(* PLC project addition_10, Dassault Systèmes ControlBuild 2024x *)
(* stored: creationDateTime 2023-10-03T11:13:32-01:00 *)

(* This module simulates the addition of maximum 10 real numbers. *)
FUNCTION_BLOCK equipment_library.addition_10
  VAR_INPUT
    in1 : REAL := 0.0;
    in2 : REAL := 0.0;
    in3 : REAL := 0.0;
    in4 : REAL := 0.0;
    in5 : REAL := 0.0;
    in6 : REAL := 0.0;
    in7 : REAL := 0.0;
    in8 : REAL := 0.0;
    in9 : REAL := 0.0;
    in10 : REAL := 0.0;
  END_VAR
  VAR_OUTPUT
    realValue : REAL := 0.0;
    dintValue : DINT := 0;
    intValue : INT := 0;
  END_VAR
  VAR
    d_locking : BOOL := false;
    v_d_locking : REAL := 0.0;
  END_VAR


ACTION C_source_code:
/* ----------------------------------------------------------------	*/
/* Type : Model of Operative Behaviour					*/
/* Category :  Toolbox							*/
/* Author : Dassault Systemes						*/
/* Update date : June 2018						*/
/* ----------------------------------------------------------------	*/
/* This module simulates the addition of maximum 10 real numbers.	*/
/* réels au maximum								*/
/* ----------------------------------------------------------------	*/

if (d_locking)
	realValue = v_d_locking; 			/* presetting of the realValue */
else
	realValue = in1+in2+in3+in4+in5+in6+in7+in8+in9+in10; /* result of the addition */

dintValue = realValue;

if ((dintValue >= -32768) && (dintValue <= 32767)) 
	intValue = dintValue ;
else 
	intValue  = 0;
END_ACTION
END_FUNCTION_BLOCK
